FUNCTION_BLOCK FB_Axis IMPLEMENTS I_UniversalMotor
VAR_OUTPUT

END_VAR
VAR	
		// =============== Axis reference =========================
	AxisRef			: AXIS_REF;				// Axis reference (process data plc/nc)
	
	//Motors data
	sMotorName	:	STRING := 'Motor';
	sUnits		:	STRING := 'mm';


	iNumberOfInstance	: SINT := 1; //numebr of currently used instance of MC_MoveVelocity
	// =============== Done signals of Halt and Reset =========
	bResetDone		: BOOL;					// Status of function block MC_Reset
	bHaltDone		: BOOL;					// Status of function block MC_Halt

	// =============== State variables ========================
	bStatusEnable	: BOOL;					// Enable feedback
	
	// =============== Motion parameters, override =====================
	lrVelocityAuto			: LREAL := 2;			// Target velocity
	lrAccelerationAuto		: LREAL := 100;			// Target acceleration
	lrDecelerationAuto		: LREAL := 100;			// Target deceleration
	lrJerkAuto				: LREAL := 100;			// Target jerk
	lrVelocityManual		: LREAL := 2;			// Target velocity
	lrAccelerationManual	: LREAL := 100;			// Target acceleration
	lrDecelerationManual	: LREAL := 100;			// Target deceleration
	lrJerkManual			: LREAL := 100;			// Target jerk
	lrOverride 				: LREAL := 100.0;		// Override 100%
	lrPosition				: LREAL := 0;			// Target Position
	mcBufferMode			: MC_BufferMode := MC_Aborting;		// buffer mode standard value
	lrDistanceToGo			: LREAL := 0; 			// distance do go for relative movement
	lrActualPosition		: LREAL; // actual postion
	
	// =============== Trigger function blocks ================
	fbTriggerHalt	: R_TRIG;				// Trigger to recognize rising edge of halt input
	fbTriggerReset	: R_TRIG;				// Trigger to recognize rising edge of reset input
	
//	// =============== Axis reference =========================
//	AxisRef			: AXIS_REF;				// Axis reference (process data plc/nc)
	
	// =============== Motion function blocks =================
	fbMcPower 		: MC_Power;				// FB for enable and override
	fbMcReset 		: MC_Reset;				// FB to reset axis
	fbMcStop 		: MC_Stop;				// FB to stop axis
	fbMcHalt		: MC_Halt;				// FB to halt axis

	fbMcMoveVelocity		: MC_MoveVelocity;		// FB to move axis (velocity movement)
	fbMcMoveAbsolute		: MC_MoveAbsolute;		// FB to move axis (absolute PTP movement)
	fbMcMoveRelative		: MC_MoveRelative;		// FB to move axis (relative PTP movement)
	fbReadActualVelocity	: MC_ReadActualVelocity; //FB to read actual velocity of axis
	fbReadActualPosition	: MC_ReadActualPosition;//FB to read actual position of axis
	
	bFirstCycle		:	BOOL := TRUE; // indicates first cycle
	iStepInit		:	INT; // step of initialization
	

	bMoveVelocity	:	BOOL; //do action 2 variable
	bMoveAbsolute	:	BOOL; //do action 3 variable
	bMoveRelative	:	BOOL; //do action 4 variable
	bStop			:	BOOL; //do action 5 variable

	iStepGeneral	:	INT; // step of main state of unit
	iStepAborting	:	INT;

	
	bManualMode		:	BOOL;
	
	
	fbAxisError		:	FB_Alarm;
	
	bCoupleable		:	BOOL;
	bHomingable		:	BOOL;
	bInitialized	:	BOOL;

	// =============== Error variables ========================
	bError			: BOOL;					// Error signal
	iErrorID		: UDINT;				// Error ID
	
END_VAR

IF bFirstCycle THEN
	bFirstCycle := FALSE;
END_IF
// cyclic
		StateMachine();
		
	// reset commands
		bMoveVelocity := FALSE;
		bMoveAbsolute := FALSE;
		bMoveRelative := FALSE;
		bStop := FALSE;
		
	// read error
		IF AxisRef.Status.Error THEN
			bError := TRUE;
			iErrorID :=  AxisRef.Status.ErrorID;
		END_IF
		
	// read pos
		fbReadActualPosition(Enable := TRUE, Axis:=AxisRef);
		lrActualPosition :=	fbReadActualPosition.Position;

	// error	
		//fbAxisError.Description := FUN_MergeStrings5(sMotorName, ' axis error number: ', UDINT_TO_STRING(iErrorID), '', '');
		//fbAxisError.Set(bError);

	// status bits
		bInitialized := iStepGeneral > 10;

METHOD Abort : BOOL // Abort axis, it will disable the power
VAR_INPUT
END_VAR
IF iStepGeneral <> 0 THEN
	iStepGeneral := -10;
END_IF
iStepInit := 0;

//Method output
	Abort := (iStepGeneral = 0);
END_METHOD

{attribute 'monitoring' := 'variable'}
PROPERTY AccelerationAuto : LREAL
GET
AccelerationAuto := lrAccelerationAuto;
END_GET
SET
lrAccelerationAuto := AccelerationAuto;
END_SET
END_PROPERTY

{attribute 'monitoring' := 'variable'}
PROPERTY AccelerationManual : LREAL
GET
AccelerationManual := lrAccelerationManual;
END_GET
SET
lrAccelerationManual := AccelerationManual;
END_SET
END_PROPERTY

{attribute 'monitoring' := 'variable'}
PROPERTY ActualPosition : LREAL
GET
ActualPosition := lrActualPosition;
END_GET
END_PROPERTY

{attribute 'monitoring' := 'variable'}
PROPERTY ActualVelocity : LREAL
GET
fbReadActualVelocity(Enable:=TRUE,Axis:=AxisRef);
ActualVelocity:=fbReadActualVelocity.ActualVelocity;
END_GET
END_PROPERTY

{attribute 'monitoring' := 'variable'}
PROPERTY AnyError : BOOL
GET
AnyError := bError;
END_GET
END_PROPERTY

PROPERTY AxisReference : AXIS_REF
GET
AxisReference := AxisRef;
END_GET
END_PROPERTY

{attribute 'monitoring' := 'variable'}
PROPERTY Buffering : BOOL // TRUE for Enable, FALSE for disable
SET
IF Buffering THEN
	mcBufferMode := MC_BlendingNext;
ELSE
	mcBufferMode := MC_Aborting;
END_IF;
END_SET
END_PROPERTY

METHOD Couple : BOOL
VAR_INPUT
END_VAR
VAR
END_VAR
END_METHOD

{attribute 'monitoring' := 'variable'}
PROPERTY Coupleable : BOOL
GET
Coupleable := bCoupleable;
END_GET
SET
bCoupleable := Coupleable;
END_SET
END_PROPERTY

{attribute 'monitoring' := 'variable'}
PROPERTY Coupled : BOOL
GET
Coupled := AxisRef.Status.Coupled;
END_GET
END_PROPERTY

{attribute 'monitoring' := 'variable'}
PROPERTY DecelerationAuto : LREAL
GET
DecelerationAuto := lrDecelerationAuto;
END_GET
SET
lrDecelerationAuto := DecelerationAuto;
END_SET
END_PROPERTY

{attribute 'monitoring' := 'variable'}
PROPERTY DecelerationManual : LREAL
GET
DecelerationManual := lrDecelerationManual;
END_GET
SET
lrDecelerationManual := DecelerationManual;
END_SET
END_PROPERTY

METHOD Decouple : BOOL
VAR_INPUT
END_VAR
VAR
END_VAR
END_METHOD

METHOD PROTECTED Enable
VAR_INPUT
	bEnable		: BOOL;
END_VAR
// =========================================================

fbMCPower(	Enable 			:= bEnable, 
			Enable_Positive	:= bEnable, 
			Enable_Negative	:= bEnable, 
			Override		:= lrOverride,
			Axis			:= AxisRef,
			Status			=> bStatusEnable);
			
IF fbMcPower.Error THEN
	bError		:= TRUE;
	iErrorID 	:= fbMcPower.ErrorID;
END_IF

AxisRef.ReadStatus();
//bMoves := AxisRef.Status.Moving;

// =========================================================
END_METHOD

{attribute 'monitoring' := 'variable'}
PROPERTY Enabled : BOOL
GET
Enabled := bStatusEnable;
END_GET
END_PROPERTY

METHOD FirstCycle : BOOL
VAR_INPUT
	//ipAlarmController	:	I_AlarmController;
	//ipHMIController		:	I_HMIController;
	sName				:	STRING;
END_VAR
THIS^.sMotorName := sName;

//THIS^.ipAlarmController := ipAlarmController;
//ipAlarmController.AppendError(fbAxisError);

//THIS^.ipHMIController := ipHMIController;
//ipHMIController.AppendMotor(THIS^);
END_METHOD

{attribute 'monitoring' := 'variable'}
PROPERTY HaltDone : BOOL
GET
HaltDone := bHaltDone;
END_GET
END_PROPERTY

METHOD Home : BOOL // Start axis homing
VAR_INPUT
END_VAR
Home := FALSE;
END_METHOD

{attribute 'monitoring' := 'variable'}
PROPERTY Homed : BOOL
GET
Homed := AxisRef.Status.Homed;
END_GET
END_PROPERTY

{attribute 'monitoring' := 'variable'}
PROPERTY Homingable : BOOL
GET
Homingable := bHomingable;
END_GET
SET
bHomingable := Homingable;
END_SET
END_PROPERTY

METHOD Init : BOOL // Initialize axis
VAR_INPUT
END_VAR
IF iStepGeneral = 0 THEN
	iStepGeneral := 10;
END_IF

//Method output
	Init := (iStepGeneral >= 20);
END_METHOD

{attribute 'monitoring' := 'variable'}
PROPERTY Initialized : BOOL
GET
Initialized := bInitialized;
END_GET
END_PROPERTY

{attribute 'monitoring' := 'variable'}
PROPERTY JerkAuto : LREAL
GET
JerkAuto := lrJerkAuto;
END_GET
SET
lrJerkAuto := JerkAuto;
END_SET
END_PROPERTY

{attribute 'monitoring' := 'variable'}
PROPERTY JerkManual : LREAL
GET
JerkManual := lrJerkManual;
END_GET
SET
lrJerkManual := JerkManual;
END_SET
END_PROPERTY

METHOD Jog : BOOL // Do action 2 request, for instance: 'Pick and place unit' change tool (additional inputs needed)
VAR_INPUT
	Distance	:	LREAL;
END_VAR
IF iStepGeneral = 30 THEN
	iStepGeneral := 100;
END_IF

bMoveRelative := TRUE;
lrDistanceToGo := Distance;

//Method output
	Jog := (iStepGeneral = 110);
END_METHOD

{attribute 'monitoring' := 'variable'}
PROPERTY ManualMode : BOOL
GET
ManualMode := bManualMode;
END_GET
SET
bManualMode := ManualMode;
END_SET
END_PROPERTY

{attribute 'monitoring' := 'variable'}
PROPERTY MotorName : STRING
GET
MotorName := sMotorName;
END_GET
SET
sMotorName := MotorName;
END_SET
END_PROPERTY

METHOD MoveAbsolute : BOOL // Do action 2 request, for instance: 'Pick and place unit' change tool (additional inputs needed)
VAR_INPUT
	Position : LREAL;
END_VAR
IF (iStepGeneral = 30) OR ((iStepGeneral = 90) AND (Position<>lrPosition)) THEN
	iStepGeneral := 80;
END_IF

bMoveAbsolute := TRUE;
lrPosition := Position;

//Method output
	MoveAbsolute := (iStepGeneral = 90);
END_METHOD

METHOD MoveRelative : BOOL // Do action 2 request, for instance: 'Pick and place unit' change tool (additional inputs needed)
VAR_INPUT
	Distance	:	LREAL;
END_VAR
IF iStepGeneral = 30 THEN
	iStepGeneral := 100;
END_IF

bMoveRelative := TRUE;
lrDistanceToGo := Distance;

//Method output
	MoveRelative := (iStepGeneral = 110);
END_METHOD

METHOD MoveVelocity : BOOL // Move the axis with constant velocity velocity, the velocity can be changed during movement 
VAR_INPUT
	lrVelocityIn	:	LREAL;
END_VAR
IF iStepGeneral = 30 THEN
	iStepGeneral := 60;
END_IF

bMoveVelocity := TRUE;
lrVelocityAuto := lrVelocityIn;

//Method output
	MoveVelocity := fbMcMoveVelocity.InVelocity;//(iStepGeneral = 70);
END_METHOD

{attribute 'monitoring' := 'variable'}
PROPERTY Override : LREAL
GET
Override := lrOverride;
END_GET
SET
lrOverride := Override;
END_SET
END_PROPERTY

METHOD Reset : BOOL
VAR_INPUT
END_VAR
fbMcHalt(			Execute	:= FALSE,
					Axis 	:= AxisRef);
fbMcMoveVelocity(	Execute	:= FALSE,
					Axis 	:= AxisRef);
fbMcMoveAbsolute(	Execute	:= FALSE,
					Axis 	:= AxisRef);
fbMcMoveRelative(	Execute	:= FALSE,
					Axis 	:= AxisRef);
IF AxisRef.Status.Error THEN
	fbMcReset(		Execute	:= TRUE,
					Axis 	:= AxisRef);
ELSE
	fbMcReset(		Execute	:= FALSE,
					Axis 	:= AxisRef);
END_IF
bError := FALSE;
iErrorID := 0;
fbAxisError.Reset();
Reset := TRUE;
END_METHOD

{attribute 'monitoring' := 'variable'}
PROPERTY ResetDone : BOOL
GET
ResetDone := bResetDone;
END_GET
END_PROPERTY

METHOD PROTECTED StateAborting : BOOL
VAR_INPUT
END_VAR
bInitialized := FALSE;
CASE iStepAborting OF
	0: 	fbMcHalt(	Execute	:= FALSE,
					Axis 	:= AxisRef);
		fbMcMoveVelocity(	Execute	:= FALSE,
							Axis 	:= AxisRef);
		fbMcMoveAbsolute(	Execute	:= FALSE,
							Axis 	:= AxisRef);
		fbMcMoveRelative(	Execute	:= FALSE,
							Axis 	:= AxisRef);
		fbMcReset(			Execute	:= FALSE,
							Axis 	:= AxisRef);
		fbMcStop(			Execute	:= FALSE,
							Axis 	:= AxisRef);					
		iStepAborting := 10;
	10:	fbMcStop(	Execute	:= TRUE,
					Axis 	:= AxisRef,
					Jerk := lrJerkAuto,
					Deceleration := lrDecelerationAuto);
		IF fbMcStop.Done THEN
			iStepAborting := 20;
		ELSIF fbMcStop.Error THEN
			bError := fbMcStop.Error;
			iErrorID := fbMcStop.ErrorID;
			iStepAborting := 20;
		END_IF
	20:	fbMcStop(	Execute	:= FALSE,
					Axis 	:= AxisRef);
		iStepAborting := 0;
		iStepGeneral := 0;
							
END_CASE
END_METHOD

METHOD PROTECTED StateHalt
VAR_INPUT
	bDriveHalt		: BOOL;					// Request stop
END_VAR
//TODO: copied from sample, finish before use
// =========================================================

IF bDriveHalt THEN
	// Move Execute FALSE
	fbMcMoveVelocity(	Execute	:= FALSE,
				Axis 	:= AxisRef);
ELSE
	// Reset done signal
	bHaltDone := FALSE;
END_IF

// Trigger
fbTriggerHalt(CLK := bDriveHalt);

IF fbTriggerHalt.Q THEN
	fbMcHalt(	Execute	:= TRUE,
				Axis 	:= AxisRef);
ELSE
	fbMcHalt(Axis := AxisRef);
END_IF

// Done / Error / Command aborted
IF fbMcHalt.Done OR fbMcHalt.Error OR fbMcHalt.CommandAborted THEN
	bError		:= fbMcHalt.Error;
	iErrorID 	:= fbMcHalt.ErrorID;
	bHaltDone 	:= fbMcHalt.Done;
	
	fbMcMoveVelocity(	Execute	:= FALSE,
				Axis 	:= AxisRef);
				
	fbMcHalt(	Execute	:= FALSE,
				Axis 	:= AxisRef);
END_IF

// =========================================================
END_METHOD

METHOD PROTECTED StateInit : BOOL //Unit is performing initialization
VAR_INPUT
END_VAR
VAR
END_VAR
//Sequence
	CASE iStepInit OF
		0: 	// reset axis
				fbMcReset(	Axis := AxisRef,
							Execute := TRUE);
			IF 
				fbMcReset.Done
			THEN
				fbMcReset(	Axis := AxisRef,
							Execute := FALSE);
				iStepInit := 10;
			ELSIF
				fbMcReset.Error 
			THEN
				bError := TRUE;
				iErrorID := fbMcReset.ErrorID;	
			END_IF
			
		10: // axis ready
			IF
				AxisRef.Status.StandStill
			THEN
				iStepInit := 100;
			END_IF

		100: // initialized
			iStepGeneral := 20;
	END_CASE
END_METHOD

METHOD PROTECTED StateMachine : BOOL // Sate machien of unit
VAR_INPUT
END_VAR

VAR
	StateAction6Done: INT;
END_VAR
//State machine						   
	CASE iStepGeneral OF
		0:  //Uninitialized
			Enable(FALSE);
			StateUninitialized();
	
		10: //Initializing - reset, power on, 
			Enable(TRUE);
			StateInit();
	
		20: //Initialized-Ready - nothing to do
			Enable(TRUE);
			StateReady();
		
		30: //Ready to start - wait for action
			Enable(TRUE);
			StateReadyToStart();
	
(*		40: //homing
			Enable(TRUE);
			StateHoming();
			
		50: //Homing done
			Enable(TRUE);
			StateHomingDone();
*)			
		60: //move velocity
			Enable(TRUE);
			StateMovingVelocity();
			
		//70: //Move Velocity done

		80: //move ptp absolute
			Enable(TRUE);
			StateMovingAbsolute(lrPosition);

		90: //move ptp absolute done
			Enable(TRUE);
			StateMovingAbsoluteDone();			
		
		100: //move relative
			Enable(TRUE);
			StateMovingRelative(lrDistanceToGo);
			
		110: //move relative done
			Enable(TRUE);
			StateMovingRelativeDone();
					
		120: //stop
			Enable(TRUE);
			StateStopping();
			
		130: //stop done
			Enable(TRUE);
			StateStoppingDone();
			
		-10: //aborting
			Enable(TRUE);
			StateAborting();
	END_CASE
END_METHOD

METHOD PROTECTED StateMovingAbsolute : BOOL // Unit is performing action 2
VAR_INPUT
	Position:	LREAL;
END_VAR
VAR_INST


END_VAR
VAR
	lrVelocity		:	LREAL;
	lrAcceleration	:	LREAL;
	lrDeceleration	:	LREAL;
	lrJerk			:	LREAL;
END_VAR
// reinitialization of FB for different position
	IF (fbMcMoveAbsolute.Position<>Position) AND fbMcMoveAbsolute.Busy THEN
			fbMcMoveAbsolute(	Axis			:= AxisRef,
								Execute			:= FALSE,
								BufferMode		:= mcBufferMode);
			fbMcMoveAbsolute.FB_INIT(TRUE,TRUE);

			//RETURN;
	END_IF

// motion parameters
IF bManualMode THEN 
	lrVelocity 		:=	lrVelocityManual;
	lrAcceleration	:=	lrAccelerationManual;
	lrDeceleration	:=	lrDecelerationManual;
	lrJerk			:=	lrJerkManual;
ELSE
	lrVelocity 		:=	lrVelocityAuto;
	lrAcceleration	:=	lrAccelerationAuto;
	lrDeceleration	:=	lrDecelerationAuto;
	lrJerk			:=	lrJerkAuto;
END_IF

// execution 
IF NOT fbMcMoveAbsolute.Error THEN // no error behavior
	fbMcMoveAbsolute(	Axis			:= AxisRef,
						Execute			:= TRUE,
						Position		:= Position,
						Velocity		:= lrVelocity,
						Acceleration	:= lrAcceleration,
						Deceleration	:= lrDeceleration,
						Jerk			:= lrJerk,
						BufferMode		:= mcBufferMode);
						
	IF fbMcMoveAbsolute.Done AND AxisRef.Status.InTargetPosition THEN
		iStepGeneral := 90;
	END_IF
	
ELSE // error behavior
		bError		:= TRUE;
		iErrorID 	:= fbMcMoveAbsolute.ErrorID;
		fbMcMoveAbsolute(	Axis			:= AxisRef,
							Execute			:= FALSE);
END_IF
END_METHOD

METHOD PROTECTED StateMovingAbsoluteDone : BOOL // Unit is performing action 2
VAR_INPUT

END_VAR
VAR_INST

END_VAR
VAR
	lrVelocity		:	LREAL;
	lrAcceleration	:	LREAL;
	lrDeceleration	:	LREAL;
	lrJerk			:	LREAL;
END_VAR
fbMcMoveAbsolute(	Axis			:= AxisRef,
					Execute			:= FALSE);
IF NOT bMoveAbsolute THEN
		iStepGeneral := 30;
END_IF
END_METHOD

METHOD PROTECTED StateMovingRelative : BOOL // Unit is performing action 2
VAR_INPUT
	Distance	:	LREAL;
END_VAR

VAR
	lrVelocity		: LREAL;
	lrAcceleration	: LREAL;
	lrDeceleration	: LREAL;
	lrJerk			: LREAL;
END_VAR
// motion parameters
IF bManualMode THEN 
	lrVelocity := lrVelocityManual;
	lrAcceleration	:=	lrAccelerationManual;
	lrDeceleration	:=	lrDecelerationManual;
	lrJerk	:=	lrJerkManual;
ELSE
	lrVelocity := lrVelocityAuto;
	lrAcceleration	:=	lrAccelerationAuto;
	lrDeceleration	:=	lrDecelerationAuto;
	lrJerk	:=	lrJerkAuto;
END_IF

//Execute
IF NOT fbMcMoveRelative.Error THEN // no error behavior
	fbMcMoveRelative(	Axis			:= AxisRef,
						Execute			:= TRUE,
						Distance		:= Distance,
						Velocity		:= lrVelocity,
						Acceleration	:= lrAcceleration,
						Deceleration	:= lrDeceleration,
						Jerk			:= lrJerkAuto);
						
	IF fbMcMoveRelative.Done THEN
		iStepGeneral := 110;
	END_IF
ELSE // error behavior
	fbMcMoveRelative(	Axis			:= AxisRef,
						Execute			:= FALSE);
END_IF
END_METHOD

METHOD PROTECTED StateMovingRelativeDone : BOOL // Unit has finished action 2, waiting for release of the request
VAR_INPUT
END_VAR
fbMcMoveRelative(	Axis			:= AxisRef,
					Execute			:= FALSE);
					
IF NOT bMoveRelative THEN
	iStepGeneral := 30;
END_IF
END_METHOD

METHOD PROTECTED StateMovingVelocity : BOOL // Unit is performing action 2
VAR_INPUT
END_VAR
VAR_INST
	mcDirection	:MC_Direction;
	lrVelocityPreviousCycle :LREAL;
END_VAR
VAR
	FB_INIT: INT;
END_VAR
IF NOT fbMcMoveVelocity.Error THEN // no error behavior
	//	Instance management - new instance of MC_MoveVelocity called to dynamical change of motion parameters 
		IF VelocityAuto <> lrVelocityPreviousCycle THEN

			//fbMcMoveVelocity.FB_INIT(TRUE,TRUE);
			fbMcMoveVelocity(	Execute 		:= FALSE,
								Axis 			:= AxisRef);
		END_IF
	

	//direction choose
		IF VelocityAuto>=0 THEN
			mcDirection := MC_Positive_Direction;
		ELSE
			mcDirection := MC_Negative_Direction;
		END_IF
	
	// move
	IF VelocityAuto=0 THEN
		fbMcHalt(	Execute 		:= TRUE,
					Deceleration	:= DecelerationAuto,
					BufferMode		:= mcBufferMode,
					Axis 			:= AxisRef,
					Jerk	 		:= lrJerkAuto);
		fbMcMoveVelocity(	Execute 		:= FALSE,
							Velocity 		:= ABS(VelocityAuto),
							Acceleration	:= AccelerationAuto,
							Deceleration	:= DecelerationAuto,
							BufferMode		:= mcBufferMode,
							Direction 		:= mcDirection,
							Axis 			:= AxisRef,
							Jerk	 		:= lrJerkAuto);
	ELSE
		fbMcHalt(	Execute 		:= FALSE,
					Deceleration	:= DecelerationAuto,
					BufferMode		:= mcBufferMode,
					Axis 			:= AxisRef,
					Jerk	 		:= lrJerkAuto);
		fbMcMoveVelocity(	Execute 		:= TRUE,
							Velocity 		:= ABS(VelocityAuto),
							Acceleration	:= AccelerationAuto,
							Deceleration	:= DecelerationAuto,
							BufferMode		:= mcBufferMode,
							Direction 		:= mcDirection,
							Axis 			:= AxisRef,
							Jerk	 		:= lrJerkAuto);
	END_IF
		lrVelocityPreviousCycle := VelocityAuto;
ELSE // error behavior
	bError		:= TRUE;
	iErrorID 	:= fbMcMoveVelocity.ErrorID;
	fbMcMoveVelocity(	Execute	:= FALSE,
						Axis 	:= AxisRef);
END_IF
END_METHOD

METHOD PROTECTED StateReady : BOOL // Unit is initialized
VAR_INPUT
END_VAR
iStepGeneral := 30;
END_METHOD

METHOD PROTECTED StateReadyToStart : BOOL // Unit is ready to start the cycle/action, in this state some preparation that are not a part of initialization can be performed
VAR_INPUT
END_VAR
END_METHOD

METHOD PROTECTED StateStopping : BOOL // Unit is performing action 2
VAR_INPUT
END_VAR

VAR
	bDriveStop: BOOL;
	iGeneralStep: INT;
END_VAR
// Move Execute FALSE
	fbMcMoveVelocity(	Execute	:= FALSE,
						Axis 	:= AxisRef);
	fbMcMoveAbsolute(	Execute	:= FALSE,
						Axis 	:= AxisRef);
	fbMcMoveRelative(	Execute	:= FALSE,
						Axis 	:= AxisRef);
// stop axis
	fbMcStop(	Axis :=	AxisRef,
				Deceleration := DecelerationAuto,
				Jerk := JerkAuto,
				Execute := TRUE);
			
// Done / Error / Command aborted
IF fbMcStop.Error THEN
	bError		:= fbMcStop.Error;
	iErrorID 	:= fbMcStop.ErrorID;
	bHaltDone 	:= fbMcStop.Done;
				
	fbMcStop(	Execute	:= FALSE,
				Axis 	:= AxisRef);
ELSIF fbMcStop.Done THEN				
	iStepGeneral := 130;
	fbMcStop(	Execute	:= FALSE,
				Axis 	:= AxisRef);
END_IF
END_METHOD

METHOD StateStoppingDone : BOOL
VAR_INPUT
END_VAR
//do something if necessary
IF NOT bStop THEN
	iStepGeneral := 30;
END_IF
END_METHOD

METHOD PROTECTED StateUninitialized : BOOL // Unit is uninitialized
VAR_INST

END_VAR
bInitialized := FALSE;
END_METHOD

METHOD Stop : BOOL // Do action 2 request, for instance: 'Pick and place unit' change tool (additional inputs needed)
VAR_INPUT
END_VAR
IF iStepGeneral >= 30 AND iStepGeneral <> 130 THEN
	iStepGeneral := 120;
END_IF
bStop := TRUE;

//Method output
	Stop := (iStepGeneral = 130);
END_METHOD

{attribute 'monitoring' := 'variable'}
PROPERTY Unit : STRING
GET
Unit := sUnits;
END_GET
SET
sUnits:=Unit;
END_SET
END_PROPERTY

{attribute 'monitoring' := 'variable'}
PROPERTY VelocityAuto : LREAL
GET
VelocityAuto := lrVelocityAuto;
END_GET
SET
lrVelocityAuto := VelocityAuto;
END_SET
END_PROPERTY

{attribute 'monitoring' := 'variable'}
PROPERTY VelocityManual : LREAL
GET
VelocityManual := lrVelocityManual;
END_GET
SET
lrVelocityManual := VelocityManual;
END_SET
END_PROPERTY

END_FUNCTION_BLOCK

(* stored: Version 1.1.0.1, ProductVersion 3.1.4024.12
   POU FB_Axis: Id {b1c6b773-afb1-48b1-9585-fb79793fcbea}, SpecialFunc None
   Folder FirstCycle: Id {fc06c3fa-c61c-4ccc-8dd3-20cdd987b489}
   Folder Properties: Id {67f3972a-0c92-4ace-86b7-93e4ddff9543}
   Folder ReferencesAndInterfaces: Id {ddae13c2-ad28-4131-bc03-36224e2e4aee}
   Folder Requests: Id {6ed435a1-8417-4c44-ad61-121451ba84e7}
   Folder StateMachine: Id {fcc53c43-6e77-4064-a95a-a65c7a758748}
   Method Abort: Id {2852b772-5f52-432a-953d-4f4ddd2dd030}
   Property AccelerationAuto: Id {2d45e029-c833-4cfe-8fc9-3983315aff02}
   Get Get: Id {819503f9-ab55-49ff-80c5-44196a2f947a}
   Set Set: Id {28ed00f5-2c54-49d4-a234-a322df85cdc5}
   Property AccelerationManual: Id {8daad240-5d4b-4e40-b144-b9d97eecd9eb}
   Get Get: Id {7f4c424a-41d9-49fa-b152-4d033144bb77}
   Set Set: Id {4be2039f-da0e-4d8f-81df-883651aa4a23}
   Property ActualPosition: Id {7c855fef-6e53-41b0-8cd1-9b1601cb0233}
   Get Get: Id {bd01480c-7250-44bb-8bc8-9f4933daea6e}
   Property ActualVelocity: Id {515a117e-930b-48f0-9f5d-1f77e06606dd}
   Get Get: Id {1f048c63-aec1-4597-a846-88b4027b5327}
   Property AnyError: Id {f284187a-c741-4215-8759-f8880c5ddf53}
   Get Get: Id {bf53deb6-05f3-450a-b3ef-8a6c0f1aba65}
   Property AxisReference: Id {271dc744-da37-4777-b2db-3a42118fdb6d}
   Get Get: Id {7b73ba97-2c72-4775-b856-62db035b798c}
   Property Buffering: Id {60921ace-a24c-459e-acbc-dff9360e539d}
   Set Set: Id {0472224e-4e3d-4ecf-b566-61969a21556e}
   Method Couple: Id {3a12de2a-6dfb-441b-a463-915ffc858d99}
   Property Coupleable: Id {2fdf449f-b235-46a9-8e3b-9e6d21f54fcd}
   Get Get: Id {3aa25d58-bc0c-43f9-97d0-e1c0de3c17f0}
   Set Set: Id {404c8f92-819b-4c72-a4e0-15e90484e651}
   Property Coupled: Id {f0ac7beb-14e5-4850-8e6d-a9c7b94bd8bc}
   Get Get: Id {fd55dd2c-789c-4213-81e3-97dd8027e29b}
   Property DecelerationAuto: Id {61bc9567-5dc8-48c5-8ced-197937a2e3ac}
   Get Get: Id {16f0ccab-738b-42b0-85bb-78088e4a90b0}
   Set Set: Id {9a7ff8c2-5fc6-419b-9365-75ec258d6e32}
   Property DecelerationManual: Id {e0e2ab52-d8fc-4af2-b8eb-5f29ef7c970a}
   Get Get: Id {10d28f29-c15c-4586-b47f-7e52bd960be9}
   Set Set: Id {8e4ee2fa-c169-4925-a639-4d7da3112c68}
   Method Decouple: Id {19883517-ad34-4ac4-a1cb-1b42e79ddbab}
   Method Enable: Id {1d3378d2-7366-4bb6-8bd3-bdf5c6e53f29}
   Property Enabled: Id {eb649819-1584-4353-a771-0a8b4094ca09}
   Get Get: Id {b7ccb800-f904-4cc6-aaea-3591cd2dd5f1}
   Method FirstCycle: Id {7eae56db-6644-4a6a-b3ea-936fee12ac6d}
   Property HaltDone: Id {0d848271-9218-4822-9b08-c02a97e24d34}
   Get Get: Id {6db5e857-7d4e-46cf-ae9f-b2a66392ab8e}
   Method Home: Id {64b4dc24-41a8-460e-8eb3-c1a224efe763}
   Property Homed: Id {12b6fc6f-f763-42af-8d62-cc394657c7e8}
   Get Get: Id {14c40c2f-689b-496a-9429-720bc9597044}
   Property Homingable: Id {3c3dd4d9-29d4-4b4c-9951-45025e28bd69}
   Get Get: Id {14985399-c90f-4a97-ac61-7cf870d02a43}
   Set Set: Id {75140c44-2c3d-42e1-8fc9-cd047d496393}
   Method Init: Id {e75a4185-3662-427d-a282-286c1934ccd0}
   Property Initialized: Id {51680044-e79f-4dda-9d81-00a0c3a694ff}
   Get Get: Id {3b5b7af2-07f3-4ff2-b1bc-5a8cb6eaffc8}
   Property JerkAuto: Id {6ed3fbb3-7af2-4c02-981d-be25d7c098ce}
   Get Get: Id {3a8866bf-778c-42a3-b68e-a5767e7e7478}
   Set Set: Id {f2acbec0-c697-437f-b7a8-4b6c29482ade}
   Property JerkManual: Id {1cf66cf4-e70e-47c9-bb41-1c8837819035}
   Get Get: Id {25471692-7538-44d9-96a0-84211de75ac4}
   Set Set: Id {d4e09893-ee9d-43bc-9ba7-f2a95af819a3}
   Method Jog: Id {b1ae246f-7d8d-4970-a598-09241e44ef50}
   Property ManualMode: Id {e4a21aac-fa03-4f40-8f05-3cd0c38d7d90}
   Get Get: Id {8f3816d3-9d18-4b9b-8bd5-2f6b21b97124}
   Set Set: Id {36f0191b-d0bc-428b-9816-655bde003a8b}
   Property MotorName: Id {5224a9a9-0eaa-4226-ab7d-1f470fcb99da}
   Get Get: Id {757261f2-c79e-4efd-bade-5fa732d58b32}
   Set Set: Id {69645a3b-7fbc-4dc5-9c7e-0a3ad360310f}
   Method MoveAbsolute: Id {57b8523b-9309-425d-b28d-1734c210a2cd}
   Method MoveRelative: Id {016bea76-89c5-4a2a-baa8-b73899e1a4c8}
   Method MoveVelocity: Id {82a51a53-501d-4422-b7bd-840ea8c35614}
   Property Override: Id {3aeff81c-e5b2-4863-862f-8105715ce54c}
   Get Get: Id {6ed74a14-6ea7-4215-8aa5-961f32bbcb6b}
   Set Set: Id {3a6410c7-e900-42d6-8afa-33b80cc67c64}
   Method Reset: Id {f228b3b9-8c6a-4610-85d7-9fce408ff2af}
   Property ResetDone: Id {6da96580-767b-492e-9d51-55b86415a6cb}
   Get Get: Id {718c740d-7b5a-4f0c-acb9-a42f5e59e0ae}
   Method StateAborting: Id {e32b4a69-133d-4bd6-946f-7e4160d9abc6}
   Method StateHalt: Id {1c0bce41-82e7-4c93-8718-33e59f4aae04}
   Method StateInit: Id {bbb82912-989d-4147-826b-729f9c2b210d}
   Method StateMachine: Id {ae1b5fd0-92be-4c31-8e76-b72847c4ef3b}
   Method StateMovingAbsolute: Id {93932c21-5015-482d-9553-320812e0a5ac}
   Method StateMovingAbsoluteDone: Id {7bd905f1-54e3-423b-9a40-17d3dac40cff}
   Method StateMovingRelative: Id {e4c97ec4-917a-4fca-a172-f3911fa3196c}
   Method StateMovingRelativeDone: Id {2be6e84d-8000-4a30-99c9-3726b55abda1}
   Method StateMovingVelocity: Id {dd4f8a5e-0ffe-467b-b7f2-9efe7d90e86c}
   Method StateReady: Id {73ea859d-52db-43fe-a713-5cec26a19312}
   Method StateReadyToStart: Id {207b3239-ffae-4782-a131-40480dd41456}
   Method StateStopping: Id {ff3086ad-7500-4875-9426-584faee6d11b}
   Method StateStoppingDone: Id {c6fd5960-4992-4dc3-ba61-1a0b43ccd17a}
   Method StateUninitialized: Id {9813e58e-617a-4670-a7c1-9d8205bbb4c2}
   Method Stop: Id {bc98f6ba-a66c-445f-a364-1b55845b95c2}
   Property Unit: Id {146f2f82-6dac-46df-b219-f12e61a4baee}
   Get Get: Id {0710f5ab-72ed-4959-bde4-49f42eb6e534}
   Set Set: Id {e581bbcf-8262-47b3-9316-f0978b0127d3}
   Property VelocityAuto: Id {17ffa7d9-8327-40bf-863c-d0194e95c548}
   Get Get: Id {56d25606-4c50-44d7-8ae0-58ad620af88d}
   Set Set: Id {5171ae62-70f3-42f1-8f74-128776b70172}
   Property VelocityManual: Id {7bffede0-1d10-4c80-9503-5cfd6ec15f11}
   Get Get: Id {7cc6b1f9-6bd5-42ad-9b0a-a27367b646f1}
   Set Set: Id {ca929778-4609-4032-b8a1-aff7b22bec13} *)
